{attribute 'GeneratedUsingTerminal: EK1100-0000-0018'}
{attribute addProperty BoxType "EK1100-0000-0018"}
{attribute addProperty Id "Term_334_EL1809EL1809_32157CFD20"}
{attribute addProperty CRC "493822018"}
{attribute addProperty Size "20"}
{attribute addProperty Name "Term 333 (EK1100)"}
TYPE Term_333_EK1100_1D6F2042 EXTENDS EK1100_1FC0878B :
STRUCT
	{attribute addProperty Name "Term 334 (EL1809)"}
	{attribute addProperty PreviousPort "Term 333 (EK1100) : B"}
	{attribute addProperty SyncUnit "default"}
	Term_334_EL1809 : EL1809_32157CFD;
END_STRUCT
END_TYPE

(* stored: Version 1.2.0.0, ProductVersion 3.1.4024.11
   DUT Term_333_EK1100_1D6F2042: Id {43dfe142-a3dc-4527-9735-ae7891b844bb} *)
